# EPICS substitutions: db/Beckhoff_5XXX/ecmcEL5101-0010.substitutions
file "ecmcEL51xx-32bit-chX.template"
{
    pattern {CH_ID}
            {01   }
}
